// TIA Portal project "MODBUS_1200_1200" (V11)

(* hardware
DEVICE "Estación SIMATIC 1200_1"  S71200.Device
   slot 0: "Rack S7-1200"  Rack  V1.0
   slot 1: "MASTER"  CPU 1214C AC/DC/Rly  6ES7 214-1BE30-0XB0  V2.2
   slot 3: "AQ1 x 12bits_1"  6ES7 232-4HA30-0XB0  V1.0
DEVICE "Estación SIMATIC 1200_2"  S71200.Device
   slot 0: "Rack S7-1200"  Rack  V1.0
   slot 1: "SLAVE"  CPU 1214C AC/DC/Rly  6ES7 214-1BE30-0XB0  V2.2
   slot 3: "AQ1 x 12bits_1"  6ES7 232-4HA30-0XB0  V1.0
*)

// ===== PLC "MASTER"  CPU 1214C AC/DC/Rly =====

VAR_GLOBAL   // PLC tag table "Tabla de variables estándar"
   "Tag_1" AT %I0.0 : Bool;
   "Tag_2" AT %I0.5 : Bool;
   "Tag_7" AT %I0.7 : Bool;
   "Tag_5" AT %MW1000 : Word;
END_VAR

ORGANIZATION_BLOCK "Main"   // OB1, LAD, ProgramCycle
TITLE = "Main Program Sweep (Cycle)"
{ S7_Optimized_Access := 'FALSE' }
VERSION : 0.1
BEGIN

REGION Network 1
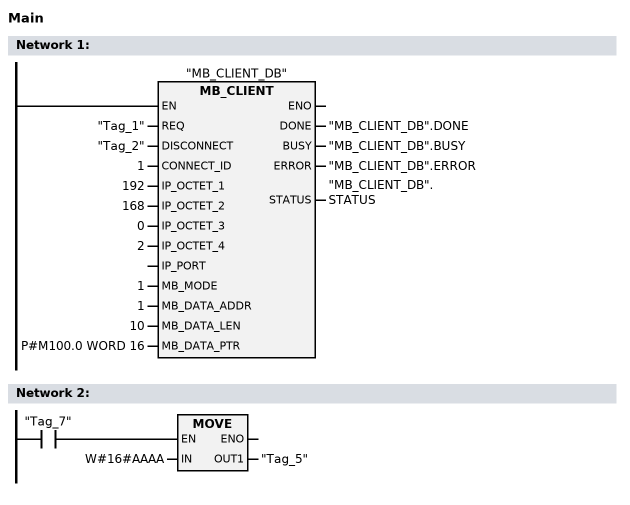
   "MB_CLIENT_DB"(REQ := "Tag_1",   // MB_CLIENT
                  DISCONNECT := "Tag_2",
                  CONNECT_ID := 1,
                  IP_OCTET_1 := 192,
                  IP_OCTET_2 := 168,
                  IP_OCTET_3 := 0,
                  IP_OCTET_4 := 2,
                  MB_MODE := 1,
                  MB_DATA_ADDR := 1,
                  MB_DATA_LEN := 10,
                  MB_DATA_PTR := P#M100.0 WORD 16,
                  DONE => "MB_CLIENT_DB".DONE,
                  BUSY => "MB_CLIENT_DB".BUSY,
                  ERROR => "MB_CLIENT_DB".ERROR,
                  STATUS => "MB_CLIENT_DB".STATUS);
END_REGION

REGION Network 2
   RUNG wire#powerrail
      Contact( "Tag_7" )
      { S7_GenerateENO := "TRUE" } Move(in := W#16#AAAA, out1 => "Tag_5")
   END_RUNG
   // the same network as SCL:
   IF "Tag_7" THEN "Tag_5" := W#16#AAAA; END_IF;
END_REGION
END_ORGANIZATION_BLOCK

// ===== PLC "SLAVE"  CPU 1214C AC/DC/Rly =====

VAR_GLOBAL   // PLC tag table "Tabla de variables estándar"
   "Tag_1" AT %I0.0 : Bool;
END_VAR

ORGANIZATION_BLOCK "Main"   // OB1, LAD, ProgramCycle
TITLE = "Main Program Sweep (Cycle)"
{ S7_Optimized_Access := 'FALSE' }
VERSION : 0.1
BEGIN

REGION Network 1
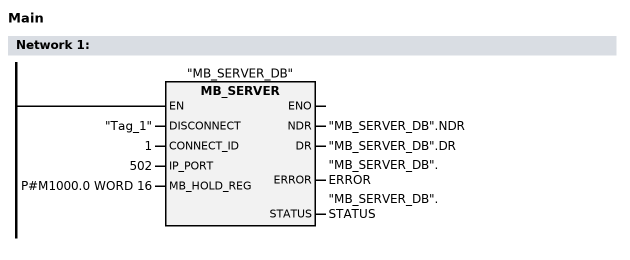
   "MB_SERVER_DB"(DISCONNECT := "Tag_1",   // MB_SERVER
                  CONNECT_ID := 1,
                  IP_PORT := 502,
                  MB_HOLD_REG := P#M1000.0 WORD 16,
                  NDR => "MB_SERVER_DB".NDR,
                  DR => "MB_SERVER_DB".DR,
                  ERROR => "MB_SERVER_DB".ERROR,
                  STATUS => "MB_SERVER_DB".STATUS);
END_REGION
END_ORGANIZATION_BLOCK